TYPE FileExtension : STRING(255);
END_TYPE

(* stored: Version 1.1.0.1, ProductVersion 3.1.4024.9
   DUT FileExtension: Id {fc84d5e5-e363-433f-ac2a-a674a888aa10} *)
